// SIMATIC S7-200 project (STEP 7-Micro/WIN), CPU 224XP REL 02.01

SYMBOL_TABLE USUARIO1
PARO_1           I0.0
PAR0_2           I0.1
MARCHA_1         I0.2
MARCHA_2         I0.3
MARCHA_3         I0.4
LAMPARA_1        Q0.0
LAMPARA_2        Q0.1
LAMPARA_3        Q0.2
END_SYMBOL_TABLE

ORGANIZATION_BLOCK PRINCIPAL:OB1
TITLE=COMENTARIOS DEL PROGRAMA
BEGIN
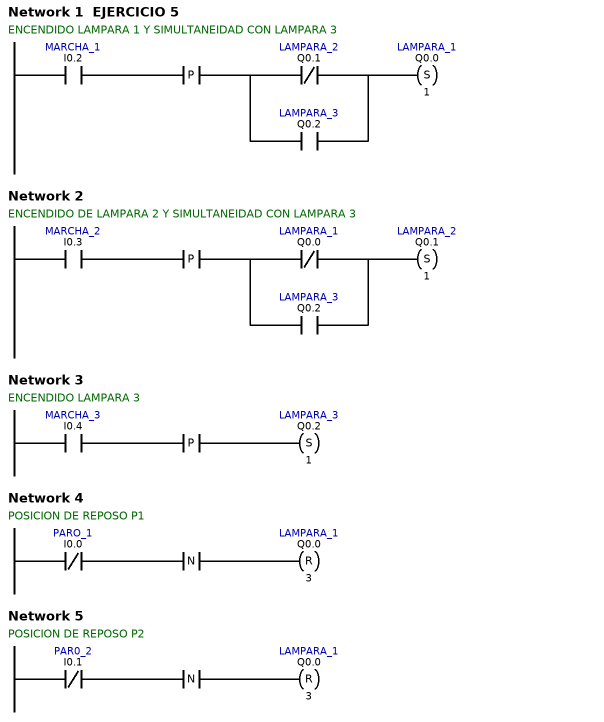
Network 1 // EJERCICIO 5
// ENCENDIDO LAMPARA 1 Y SIMULTANEIDAD CON LAMPARA 3
LD     MARCHA_1:I0.2
EU
LDN    LAMPARA_2:Q0.1
O      LAMPARA_3:Q0.2
ALD
S      LAMPARA_1:Q0.0, 1
Network 2
// ENCENDIDO DE LAMPARA 2 Y SIMULTANEIDAD CON LAMPARA 3
LD     MARCHA_2:I0.3
EU
LDN    LAMPARA_1:Q0.0
O      LAMPARA_3:Q0.2
ALD
S      LAMPARA_2:Q0.1, 1
Network 3
// ENCENDIDO LAMPARA 3 
LD     MARCHA_3:I0.4
EU
S      LAMPARA_3:Q0.2, 1
Network 4
// POSICION DE REPOSO P1
LDN    PARO_1:I0.0
ED
R      LAMPARA_1:Q0.0, 3
Network 5
// POSICION DE REPOSO P2
LDN    PAR0_2:I0.1
ED
R      LAMPARA_1:Q0.0, 3
END_ORGANIZATION_BLOCK
